  MoveL 9737 to (-47.88, -48.32, -15.5) mm, rotated rx 180 ry 0 rz 90 deg; joints [71.765, -17.653, 86.431, 0, 21.222, 71.765]
  Establecer velocidad (1000.0 mm/s)
  MoveL 9738 to (-47.88, -48.32, 10) mm, rotated rx 180 ry 0 rz 90 deg; joints [71.765, -18.97, 87.289, 0, 21.68, 71.765]
  Establecer velocidad (66.7 mm/s)
  MoveL 9739 to (-51.43, -54.96, 10) mm, rotated rx 180 ry 0 rz 90 deg; joints [71.511, -18.993, 87.381, 0, 21.611, 71.511]
  MoveL 9740 to (-51.43, -54.96, -15.5) mm, rotated rx -180 ry 0 rz 90 deg; joints [71.511, -17.675, 86.523, 0, 21.152, 71.511]
  MoveL 9741 to (-49.93, -55.15, -15.91) mm, rotated rx -180 ry 0 rz 90 deg; joints [71.521, -17.628, 86.402, 0, 21.226, 71.521]
  MoveL 9742 to (-48.42, -54.96, -16.31) mm, rotated rx -180 ry 0 rz 90 deg; joints [71.544, -17.583, 86.289, 0, 21.294, 71.544]
  MoveL 9743 to (-46.99, -54.45, -16.72) mm, rotated rx 180 ry 0 rz 90 deg; joints [71.576, -17.541, 86.189, 0, 21.352, 71.576]
  MoveL 9744 to (-45.7, -53.64, -17.12) mm, rotated rx 180 ry 0 rz 90 deg; joints [71.616, -17.504, 86.106, 0, 21.398, 71.616]
  MoveL 9745 to (-44.64, -52.56, -17.53) mm, rotated rx 180 ry 0 rz 90 deg; joints [71.663, -17.471, 86.043, 0, 21.428, 71.663]
  MoveL 9746 to (-43.83, -51.27, -17.94) mm, rotated rx -180 ry 0 rz 90 deg; joints [71.713, -17.443, 86.003, 0, 21.44, 71.713]
  MoveL 9747 to (-43.33, -49.83, -18.34) mm, rotated rx 180 ry 0 rz 90 deg; joints [71.765, -17.422, 85.987, 0, 21.435, 71.765]
  MoveL 9748 to (-43.19, -48.32, -18.75) mm, rotated rx -180 ry 0 rz 90 deg; joints [71.816, -17.407, 85.998, 0, 21.409, 71.816]
  MoveL 9749 to (-43.19, -30.36, -18.75) mm, rotated rx -180 ry 0 rz 90 deg; joints [72.401, -17.503, 86.396, 0, 21.108, 72.401]
  MoveL 9750 to (-45.96, -30.86, -18.75) mm, rotated rx -180 ry 0 rz 90 deg; joints [72.356, -17.546, 86.574, 0, 20.972, 72.356]
  MoveL 9751 to (-62.07, -33.84, -18.75) mm, rotated rx -180 ry 0 rz 90 deg; joints [72.088, -17.79, 87.605, 0, 20.185, 72.088]
  MoveL 9752 to (-65.86, -34.57, -18.75) mm, rotated rx 180 ry 0 rz 90 deg; joints [72.024, -17.845, 87.845, 0, 20.001, 72.024]
  MoveC 9753 to (-67.04, -35.24, -18.75) mm, rotated rx -180 ry 0 rz 90 deg; joints [71.989, -17.86, 87.909, 0, 19.951, 71.989] to (-67.55, -36.48, -18.75) mm, rotated rx 180 ry 0 rz 90 deg; joints [71.942, -17.862, 87.917, 0, 19.945, 71.942]
  MoveL 9754 to (-67.58, -36.96, -18.75) mm, rotated rx 180 ry 0 rz 90 deg; joints [71.926, -17.86, 87.908, 0, 19.952, 71.926]
  MoveL 9755 to (-67.57, -65.53, -18.75) mm, rotated rx 180 ry 0 rz 90 deg; joints [70.987, -17.71, 87.262, 0, 20.447, 70.987]
  MoveC 9756 to (-66.92, -67.07, -18.75) mm, rotated rx -180 ry 0 rz 90 deg; joints [70.944, -17.691, 87.182, 0, 20.509, 70.944] to (-65.35, -67.68, -18.75) mm, rotated rx -180 ry 0 rz 90 deg; joints [70.942, -17.663, 87.062, 0, 20.6, 70.942]
  MoveC 9757 to (-54.27, -67.34, -18.75) mm, rotated rx 180 ry 0 rz 90 deg; joints [71.077, -17.485, 86.319, 0, 21.166, 71.077] to (-43.19, -66.92, -18.75) mm, rotated rx 180 ry 0 rz 90 deg; joints [71.213, -17.302, 85.571, 0, 21.731, 71.213]
  MoveL 9758 to (-43.19, -48.32, -18.75) mm, rotated rx -180 ry 0 rz 90 deg; joints [71.816, -17.407, 85.998, 0, 21.409, 71.816]
  MoveL 9759 to (-50.74, -48.32, -18.75) mm, rotated rx -180 ry 0 rz 90 deg; joints [71.735, -17.532, 86.514, 0, 21.018, 71.735]
  MoveL 9760 to (-50.74, -48.32, -15.75) mm, rotated rx 180 ry 0 rz 90 deg; joints [71.735, -17.687, 86.618, 0, 21.069, 71.735]
  Establecer velocidad (1000.0 mm/s)
  MoveL 9761 to (-50.74, -48.32, 10) mm, rotated rx 180 ry 0 rz 90 deg; joints [71.735, -19.018, 87.485, 0, 21.534, 71.735]
  Establecer velocidad (66.7 mm/s)
  MoveL 9762 to (-59.34, 34.85, 10) mm, rotated rx 180 ry 0 rz 90 deg; joints [74.408, -19.568, 89.788, 0, 19.78, 74.408]
  MoveL 9763 to (-59.34, 34.85, -15.5) mm, rotated rx 180 ry 0 rz 90 deg; joints [74.408, -18.236, 88.929, 0, 19.307, 74.408]
  MoveL 9764 to (-60.84, 35.03, -15.91) mm, rotated rx 180 ry 0 rz 90 deg; joints [74.4, -18.238, 89.02, 0, 19.218, 74.4]
  MoveL 9765 to (-62.35, 34.85, -16.31) mm, rotated rx 180 ry 0 rz 90 deg; joints [74.38, -18.239, 89.104, 0, 19.135, 74.38]
  MoveL 9766 to (-63.78, 34.34, -16.72) mm, rotated rx 180 ry 0 rz 90 deg; joints [74.349, -18.237, 89.177, 0, 19.06, 74.349]
  MoveL 9767 to (-65.06, 33.52, -17.12) mm, rotated rx -180 ry 0 rz 90 deg; joints [74.309, -18.231, 89.234, 0, 18.997, 74.309]
  MoveL 9768 to (-66.13, 32.44, -17.53) mm, rotated rx -180 ry 0 rz 90 deg; joints [74.262, -18.221, 89.271, 0, 18.95, 74.262]
  MoveL 9769 to (-66.94, 31.15, -17.94) mm, rotated rx 180 ry 0 rz 90 deg; joints [74.211, -18.207, 89.287, 0, 18.92, 74.211]
  MoveL 9770 to (-67.44, 29.72, -18.34) mm, rotated rx 180 ry 0 rz 90 deg; joints [74.158, -18.187, 89.279, 0, 18.907, 74.158]
  MoveL 9771 to (-67.58, 28.21, -18.75) mm, rotated rx 180 ry 0 rz 90 deg; joints [74.105, -18.161, 89.246, 0, 18.915, 74.105]
  MoveL 9772 to (-67.58, 7.58, -18.75) mm, rotated rx 180 ry 0 rz 90 deg; joints [73.41, -18.072, 88.842, 0, 19.229, 73.41]
  MoveL 9773 to (-67.56, 7.11, -18.75) mm, rotated rx 180 ry 0 rz 90 deg; joints [73.394, -18.069, 88.832, 0, 19.237, 73.394]
  MoveC 9774 to (-66.64, 5.61, -18.75) mm, rotated rx 180 ry 0 rz 90 deg; joints [73.354, -18.049, 88.74, 0, 19.309, 73.354] to (-64.91, 5.24, -18.75) mm, rotated rx 180 ry 0 rz 90 deg; joints [73.358, -18.021, 88.616, 0, 19.405, 73.358]
  MoveL 9775 to (-63.02, 5.72, -18.75) mm, rotated rx 180 ry 0 rz 90 deg; joints [73.393, -17.994, 88.498, 0, 19.496, 73.393]
  MoveL 9776 to (-45.01, 10.34, -18.75) mm, rotated rx 180 ry 0 rz 90 deg; joints [73.724, -17.735, 87.369, 0, 20.366, 73.724]
  MoveL 9777 to (-43.19, 10.83, -18.75) mm, rotated rx 180 ry 0 rz 90 deg; joints [73.758, -17.708, 87.254, 0, 20.454, 73.758]
  MoveL 9778 to (-43.19, 36.65, -18.75) mm, rotated rx 180 ry 0 rz 90 deg; joints [74.619, -17.824, 87.754, 0, 20.07, 74.619]
  MoveC 9779 to (-53.63, 43.7, -18.75) mm, rotated rx 180 ry 0 rz 90 deg; joints [74.76, -18.017, 88.596, 0, 19.42, 74.76] to (-64.1, 50.7, -18.75) mm, rotated rx 180 ry 0 rz 90 deg; joints [74.901, -18.202, 89.431, 0, 18.771, 74.901]
  MoveC 9780 to (-64.36, 50.84, -18.75) mm, rotated rx -180 ry 0 rz 90 deg; joints [74.903, -18.206, 89.451, 0, 18.755, 74.903] to (-64.66, 50.91, -18.75) mm, rotated rx 180 ry 0 rz 90 deg; joints [74.903, -18.211, 89.472, 0, 18.739, 74.903]
  MoveC 9781 to (-66.38, 50.6, -18.75) mm, rotated rx 180 ry 0 rz 90 deg; joints [74.876, -18.235, 89.583, 0, 18.652, 74.876] to (-67.57, 49.31, -18.75) mm, rotated rx 180 ry 0 rz 90 deg; joints [74.822, -18.247, 89.639, 0, 18.608, 74.822]
  MoveL 9782 to (-67.58, 48.8, -18.75) mm, rotated rx -180 ry 0 rz 90 deg; joints [74.804, -18.245, 89.63, 0, 18.615, 74.804]
  MoveL 9783 to (-67.58, 28.21, -18.75) mm, rotated rx 180 ry 0 rz 90 deg; joints [74.105, -18.161, 89.246, 0, 18.915, 74.105]
  MoveL 9784 to (-60.03, 28.21, -18.75) mm, rotated rx -180 ry 0 rz 90 deg; joints [74.178, -18.048, 88.738, 0, 19.311, 74.178]
  MoveL 9785 to (-60.03, 28.21, -15.75) mm, rotated rx 180 ry 0 rz 90 deg; joints [74.178, -18.205, 88.841, 0, 19.364, 74.178]
  Establecer velocidad (1000.0 mm/s)
  MoveL 9786 to (-60.03, 28.21, 10) mm, rotated rx -180 ry 0 rz 90 deg; joints [74.178, -19.549, 89.708, 0, 19.841, 74.178]
  Establecer velocidad (66.7 mm/s)
  MoveL 9787 to (-59.17, 34.85, 10) mm, rotated rx 180 ry 0 rz 90 deg; joints [74.41, -19.565, 89.777, 0, 19.789, 74.41]
  MoveL 9788 to (-59.17, 34.85, -15.75) mm, rotated rx 180 ry 0 rz 90 deg; joints [74.41, -18.22, 88.909, 0, 19.311, 74.41]
  MoveL 9789 to (-60.68, 35.03, -16.16) mm, rotated rx 180 ry 0 rz 90 deg; joints [74.402, -18.223, 89, 0, 19.222, 74.402]
  MoveL 9790 to (-62.19, 34.85, -16.56) mm, rotated rx 180 ry 0 rz 90 deg; joints [74.381, -18.223, 89.085, 0, 19.139, 74.381]
  MoveL 9791 to (-63.62, 34.34, -16.97) mm, rotated rx -180 ry 0 rz 90 deg; joints [74.351, -18.221, 89.158, 0, 19.064, 74.351]
  MoveL 9792 to (-64.9, 33.52, -17.38) mm, rotated rx 180 ry 0 rz 90 deg; joints [74.311, -18.216, 89.214, 0, 19.002, 74.311]
  MoveL 9793 to (-65.97, 32.44, -17.78) mm, rotated rx 180 ry 0 rz 90 deg; joints [74.264, -18.206, 89.252, 0, 18.954, 74.264]
  MoveL 9794 to (-66.77, 31.15, -18.19) mm, rotated rx 180 ry 0 rz 90 deg; joints [74.213, -18.191, 89.267, 0, 18.924, 74.213]
  MoveL 9795 to (-67.27, 29.72, -18.59) mm, rotated rx 180 ry 0 rz 90 deg; joints [74.159, -18.171, 89.26, 0, 18.912, 74.159]
  MoveL 9796 to (-67.41, 28.21, -19) mm, rotated rx 180 ry 0 rz 90 deg; joints [74.107, -18.146, 89.226, 0, 18.92, 74.107]
  MoveL 9797 to (-67.41, 7.58, -19) mm, rotated rx 180 ry 0 rz 90 deg; joints [73.412, -18.056, 88.823, 0, 19.234, 73.412]
  MoveC 9798 to (-66.67, 5.91, -19) mm, rotated rx 180 ry 0 rz 90 deg; joints [73.363, -18.038, 88.739, 0, 19.298, 73.363] to (-64.91, 5.4, -19) mm, rotated rx 180 ry 0 rz 90 deg; joints [73.364, -18.009, 88.611, 0, 19.398, 73.364]
  MoveL 9799 to (-64.44, 5.5, -19) mm, rotated rx -180 ry 0 rz 90 deg; joints [73.372, -18.002, 88.581, 0, 19.421, 73.372]
  MoveL 9800 to (-61.12, 6.33, -19) mm, rotated rx 180 ry 0 rz 90 deg; joints [73.433, -17.955, 88.374, 0, 19.581, 73.433]
  MoveL 9801 to (-46.91, 10, -19) mm, rotated rx 180 ry 0 rz 90 deg; joints [73.695, -17.75, 87.483, 0, 20.267, 73.695]
  MoveL 9802 to (-46.05, 10.22, -19) mm, rotated rx 180 ry 0 rz 90 deg; joints [73.711, -17.738, 87.429, 0, 20.309, 73.711]
  MoveL 9803 to (-46.05, 38.41, -19) mm, rotated rx -180 ry 0 rz 90 deg; joints [74.652, -17.864, 87.974, 0, 19.89, 74.652]
  MoveC 9804 to (-55.14, 44.54, -19) mm, rotated rx 180 ry 0 rz 90 deg; joints [74.775, -18.03, 88.705, 0, 19.325, 74.775] to (-64.26, 50.63, -19) mm, rotated rx -180 ry 0 rz 90 deg; joints [74.897, -18.191, 89.432, 0, 18.759, 74.897]
  MoveC 9805 to (-66.11, 50.42, -19) mm, rotated rx 180 ry 0 rz 90 deg; joints [74.873, -18.217, 89.552, 0, 18.665, 74.873] to (-67.41, 49.08, -19) mm, rotated rx -180 ry 0 rz 90 deg; joints [74.815, -18.231, 89.615, 0, 18.616, 74.815]
  MoveL 9806 to (-67.41, 48.8, -19) mm, rotated rx -180 ry 0 rz 90 deg; joints [74.806, -18.23, 89.611, 0, 18.619, 74.806]
  MoveL 9807 to (-67.41, 28.21, -19) mm, rotated rx 180 ry 0 rz 90 deg; joints [74.107, -18.146, 89.226, 0, 18.92, 74.107]
  MoveL 9808 to (-59.86, 28.21, -19) mm, rotated rx 180 ry 0 rz 90 deg; joints [74.179, -18.033, 88.718, 0, 19.315, 74.179]
  MoveL 9809 to (-59.86, 28.21, -16) mm, rotated rx 180 ry 0 rz 90 deg; joints [74.179, -18.19, 88.821, 0, 19.368, 74.179]
  Establecer velocidad (1000.0 mm/s)
  MoveL 9810 to (-59.86, 28.21, 10) mm, rotated rx 180 ry 0 rz 90 deg; joints [74.179, -19.547, 89.697, 0, 19.85, 74.179]
  Establecer velocidad (66.7 mm/s)
  MoveL 9811 to (-59.17, -44.43, 10) mm, rotated rx -180 ry 0 rz 90 deg; joints [71.771, -19.18, 88.145, 0, 21.035, 71.771]
  MoveL 9812 to (-59.17, -44.43, -15.75) mm, rotated rx 180 ry 0 rz 90 deg; joints [71.771, -17.845, 87.278, 0, 20.567, 71.771]
  MoveL 9813 to (-60.68, -44.25, -16.16) mm, rotated rx 180 ry 0 rz 90 deg; joints [71.761, -17.849, 87.37, 0, 20.478, 71.761]
  MoveL 9814 to (-62.19, -44.43, -16.56) mm, rotated rx 180 ry 0 rz 90 deg; joints [71.738, -17.851, 87.454, 0, 20.396, 71.738]
  MoveL 9815 to (-63.62, -44.94, -16.97) mm, rotated rx 180 ry 0 rz 90 deg; joints [71.706, -17.85, 87.526, 0, 20.324, 71.706]
  MoveL 9816 to (-64.9, -45.76, -17.38) mm, rotated rx -180 ry 0 rz 90 deg; joints [71.665, -17.844, 87.58, 0, 20.264, 71.665]
  MoveL 9817 to (-65.97, -46.84, -17.78) mm, rotated rx -180 ry 0 rz 90 deg; joints [71.618, -17.835, 87.614, 0, 20.221, 71.618]
  MoveL 9818 to (-66.77, -48.13, -18.19) mm, rotated rx -180 ry 0 rz 90 deg; joints [71.567, -17.819, 87.625, 0, 20.194, 71.567]
  MoveL 9819 to (-67.27, -49.56, -18.59) mm, rotated rx -180 ry 0 rz 90 deg; joints [71.514, -17.798, 87.613, 0, 20.186, 71.514]
  MoveL 9820 to (-67.41, -51.07, -19) mm, rotated rx 180 ry 0 rz 90 deg; joints [71.463, -17.772, 87.574, 0, 20.198, 71.463]
  MoveL 9821 to (-67.41, -64.91, -19) mm, rotated rx 180 ry 0 rz 90 deg; joints [71.009, -17.698, 87.257, 0, 20.44, 71.009]
  MoveL 9822 to (-67.41, -65.39, -19) mm, rotated rx -180 ry 0 rz 90 deg; joints [70.994, -17.695, 87.246, 0, 20.449, 70.994]
  MoveC 9823 to (-66.84, -66.87, -19) mm, rotated rx 180 ry 0 rz 90 deg; joints [70.952, -17.678, 87.173, 0, 20.505, 70.952] to (-65.39, -67.53, -19) mm, rotated rx -180 ry 0 rz 90 deg; joints [70.947, -17.651, 87.06, 0, 20.591, 70.947]
  MoveL 9824 to (-64.91, -67.53, -19) mm, rotated rx 180 ry 0 rz 90 deg; joints [70.952, -17.643, 87.028, 0, 20.616, 70.952]
  MoveL 9825 to (-47.86, -66.96, -19) mm, rotated rx -180 ry 0 rz 90 deg; joints [71.161, -17.368, 85.881, 0, 21.486, 71.161]
  MoveL 9826 to (-46.05, -66.87, -19) mm, rotated rx -180 ry 0 rz 90 deg; joints [71.183, -17.338, 85.759, 0, 21.578, 71.183]
  MoveL 9827 to (-46.05, -31.04, -19) mm, rotated rx -180 ry 0 rz 90 deg; joints [72.349, -17.534, 86.568, 0, 20.966, 72.349]
  MoveL 9828 to (-62.07, -34, -19) mm, rotated rx 180 ry 0 rz 90 deg; joints [72.083, -17.776, 87.593, 0, 20.183, 72.083]
  MoveL 9829 to (-65.71, -34.69, -19) mm, rotated rx -180 ry 0 rz 90 deg; joints [72.021, -17.829, 87.823, 0, 20.006, 72.021]
  MoveC 9830 to (-66.93, -35.42, -19) mm, rotated rx 180 ry 0 rz 90 deg; joints [71.984, -17.845, 87.89, 0, 19.955, 71.984] to (-67.41, -36.76, -19) mm, rotated rx -180 ry 0 rz 90 deg; joints [71.935, -17.845, 87.893, 0, 19.953, 71.935]
  MoveL 9831 to (-67.41, -51.07, -19) mm, rotated rx 180 ry 0 rz 90 deg; joints [71.463, -17.772, 87.574, 0, 20.198, 71.463]
  MoveL 9832 to (-59.86, -51.07, -19) mm, rotated rx -180 ry 0 rz 90 deg; joints [71.546, -17.652, 87.064, 0, 20.588, 71.546]
  MoveL 9833 to (-59.86, -51.07, -16) mm, rotated rx 180 ry 0 rz 90 deg; joints [71.546, -17.808, 87.167, 0, 20.64, 71.546]
  Establecer velocidad (1000.0 mm/s)
  MoveL 9834 to (-59.86, -51.07, 10) mm, rotated rx -180 ry 0 rz 90 deg; joints [71.546, -19.155, 88.042, 0, 21.112, 71.546]
  Establecer velocidad (66.7 mm/s)
  MoveL 9835 to (-59.01, -44.43, 10) mm, rotated rx 180 ry 0 rz 90 deg; joints [71.773, -19.177, 88.134, 0, 21.043, 71.773]
  MoveL 9836 to (-59.01, -44.43, -16) mm, rotated rx 180 ry 0 rz 90 deg; joints [71.773, -17.829, 87.259, 0, 20.571, 71.773]
  MoveL 9837 to (-60.51, -44.25, -16.41) mm, rotated rx 180 ry 0 rz 90 deg; joints [71.762, -17.833, 87.351, 0, 20.483, 71.762]
  MoveL 9838 to (-62.02, -44.43, -16.81) mm, rotated rx 180 ry 0 rz 90 deg; joints [71.74, -17.835, 87.435, 0, 20.401, 71.74]
  MoveL 9839 to (-63.45, -44.94, -17.22) mm, rotated rx -180 ry 0 rz 90 deg; joints [71.708, -17.834, 87.506, 0, 20.328, 71.708]
  MoveL 9840 to (-64.73, -45.76, -17.63) mm, rotated rx -180 ry 0 rz 90 deg; joints [71.667, -17.829, 87.56, 0, 20.269, 71.667]
  MoveL 9841 to (-65.81, -46.84, -18.03) mm, rotated rx 180 ry 0 rz 90 deg; joints [71.62, -17.819, 87.594, 0, 20.225, 71.62]
  MoveL 9842 to (-66.61, -48.13, -18.44) mm, rotated rx -180 ry 0 rz 90 deg; joints [71.569, -17.804, 87.605, 0, 20.198, 71.569]
  MoveL 9843 to (-67.11, -49.56, -18.84) mm, rotated rx -180 ry 0 rz 90 deg; joints [71.516, -17.783, 87.593, 0, 20.19, 71.516]
  MoveL 9844 to (-67.25, -51.07, -19.25) mm, rotated rx 180 ry 0 rz 90 deg; joints [71.465, -17.756, 87.554, 0, 20.202, 71.465]
  MoveL 9845 to (-67.25, -65.29, -19.25) mm, rotated rx -180 ry 0 rz 90 deg; joints [70.999, -17.68, 87.229, 0, 20.451, 70.999]
  MoveC 9846 to (-66.61, -66.8, -19.25) mm, rotated rx 180 ry 0 rz 90 deg; joints [70.957, -17.661, 87.15, 0, 20.511, 70.957] to (-65.07, -67.4, -19.25) mm, rotated rx -180 ry 0 rz 90 deg; joints [70.955, -17.634, 87.033, 0, 20.601, 70.955]
  MoveL 9847 to (-63.02, -67.33, -19.25) mm, rotated rx 180 ry 0 rz 90 deg; joints [70.98, -17.601, 86.895, 0, 20.706, 70.98]
  MoveL 9848 to (-51.65, -66.94, -19.25) mm, rotated rx -180 ry 0 rz 90 deg; joints [71.119, -17.418, 86.132, 0, 21.286, 71.119]
  MoveL 9849 to (-48.91, -66.84, -19.25) mm, rotated rx -180 ry 0 rz 90 deg; joints [71.153, -17.373, 85.947, 0, 21.426, 71.153]
  MoveL 9850 to (-48.91, -31.73, -19.25) mm, rotated rx 180 ry 0 rz 90 deg; joints [72.297, -17.564, 86.74, 0, 20.824, 72.297]
  MoveL 9851 to (-51.65, -32.22, -19.25) mm, rotated rx -180 ry 0 rz 90 deg; joints [72.252, -17.606, 86.916, 0, 20.69, 72.252]
  MoveL 9852 to (-65.58, -34.82, -19.25) mm, rotated rx 180 ry 0 rz 90 deg; joints [72.019, -17.814, 87.803, 0, 20.011, 72.019]
  MoveC 9853 to (-66.78, -35.52, -19.25) mm, rotated rx 180 ry 0 rz 90 deg; joints [71.983, -17.829, 87.868, 0, 19.961, 71.983] to (-67.25, -36.82, -19.25) mm, rotated rx -180 ry 0 rz 90 deg; joints [71.934, -17.829, 87.871, 0, 19.958, 71.934]
  MoveL 9854 to (-67.25, -51.07, -19.25) mm, rotated rx 180 ry 0 rz 90 deg; joints [71.465, -17.756, 87.554, 0, 20.202, 71.465]
  MoveL 9855 to (-59.7, -51.07, -19.25) mm, rotated rx -180 ry 0 rz 90 deg; joints [71.548, -17.636, 87.044, 0, 20.592, 71.548]
  MoveL 9856 to (-59.7, -51.07, -16.25) mm, rotated rx 180 ry 0 rz 90 deg; joints [71.548, -17.792, 87.147, 0, 20.645, 71.548]
  Establecer velocidad (1000.0 mm/s)
  MoveL 9857 to (-59.7, -51.07, 10) mm, rotated rx 180 ry 0 rz 90 deg; joints [71.548, -19.152, 88.031, 0, 21.121, 71.548]
  Establecer velocidad (66.7 mm/s)
  MoveL 9858 to (-59.01, 34.87, 10) mm, rotated rx -180 ry 0 rz 90 deg; joints [74.412, -19.563, 89.766, 0, 19.797, 74.412]
  MoveL 9859 to (-59.01, 34.87, -16) mm, rotated rx 180 ry 0 rz 90 deg; joints [74.412, -18.205, 88.89, 0, 19.315, 74.412]
  MoveL 9860 to (-60.52, 35.05, -16.41) mm, rotated rx 180 ry 0 rz 90 deg; joints [74.404, -18.207, 88.981, 0, 19.226, 74.404]
  MoveL 9861 to (-62.02, 34.87, -16.81) mm, rotated rx -180 ry 0 rz 90 deg; joints [74.384, -18.208, 89.066, 0, 19.142, 74.384]
  MoveL 9862 to (-63.45, 34.36, -17.22) mm, rotated rx -180 ry 0 rz 90 deg; joints [74.353, -18.206, 89.138, 0, 19.068, 74.353]
  MoveL 9863 to (-64.74, 33.54, -17.63) mm, rotated rx 180 ry 0 rz 90 deg; joints [74.313, -18.2, 89.195, 0, 19.005, 74.313]
  MoveL 9864 to (-65.81, 32.46, -18.03) mm, rotated rx -180 ry 0 rz 90 deg; joints [74.266, -18.19, 89.233, 0, 18.958, 74.266]
  MoveL 9865 to (-66.61, 31.18, -18.44) mm, rotated rx -180 ry 0 rz 90 deg; joints [74.215, -18.176, 89.248, 0, 18.927, 74.215]
  MoveL 9866 to (-67.11, 29.74, -18.84) mm, rotated rx 180 ry 0 rz 90 deg; joints [74.162, -18.156, 89.24, 0, 18.915, 74.162]
  MoveL 9867 to (-67.25, 28.23, -19.25) mm, rotated rx -180 ry 0 rz 90 deg; joints [74.109, -18.13, 89.207, 0, 18.923, 74.109]
  MoveL 9868 to (-67.25, 8.05, -19.25) mm, rotated rx 180 ry 0 rz 90 deg; joints [73.429, -18.043, 88.812, 0, 19.23, 73.429]
  MoveL 9869 to (-67.25, 7.58, -19.25) mm, rotated rx 180 ry 0 rz 90 deg; joints [73.414, -18.041, 88.803, 0, 19.238, 73.414]
  MoveC 9870 to (-66.51, 6.08, -19.25) mm, rotated rx 180 ry 0 rz 90 deg; joints [73.37, -18.023, 88.723, 0, 19.3, 73.37] to (-64.91, 5.55, -19.25) mm, rotated rx 180 ry 0 rz 90 deg; joints [73.369, -17.996, 88.605, 0, 19.391, 73.369]
  MoveL 9871 to (-64.44, 5.64, -19.25) mm, rotated rx 180 ry 0 rz 90 deg; joints [73.377, -17.99, 88.575, 0, 19.414, 73.377]
  MoveL 9872 to (-48.91, 9.64, -19.25) mm, rotated rx -180 ry 0 rz 90 deg; joints [73.663, -17.767, 87.603, 0, 20.164, 73.663]
  MoveL 9873 to (-48.91, 40.16, -19.25) mm, rotated rx 180 ry 0 rz 90 deg; joints [74.684, -17.903, 88.192, 0, 19.71, 74.684]
  MoveL 9874 to (-60.32, 47.86, -19.25) mm, rotated rx 180 ry 0 rz 90 deg; joints [74.839, -18.108, 89.107, 0, 19.001, 74.839]
  MoveL 9875 to (-63.15, 49.75, -19.25) mm, rotated rx 180 ry 0 rz 90 deg; joints [74.877, -18.158, 89.333, 0, 18.825, 74.877]
  MoveL 9876 to (-63.97, 50.3, -19.25) mm, rotated rx -180 ry 0 rz 90 deg; joints [74.888, -18.172, 89.398, 0, 18.775, 74.888]
  MoveL 9877 to (-64.12, 50.38, -19.25) mm, rotated rx 180 ry 0 rz 90 deg; joints [74.89, -18.175, 89.41, 0, 18.765, 74.89]
  MoveC 9878 to (-65.95, 50.18, -19.25) mm, rotated rx 180 ry 0 rz 90 deg; joints [74.866, -18.201, 89.528, 0, 18.672, 74.866] to (-67.24, 48.88, -19.25) mm, rotated rx -180 ry 0 rz 90 deg; joints [74.81, -18.214, 89.592, 0, 18.623, 74.81]
  MoveL 9879 to (-67.25, 48.8, -19.25) mm, rotated rx -180 ry 0 rz 90 deg; joints [74.807, -18.214, 89.591, 0, 18.623, 74.807]
  MoveL 9880 to (-67.25, 28.23, -19.25) mm, rotated rx -180 ry 0 rz 90 deg; joints [74.109, -18.13, 89.207, 0, 18.923, 74.109]
  MoveL 9881 to (-59.7, 28.23, -19.25) mm, rotated rx -180 ry 0 rz 90 deg; joints [74.182, -18.017, 88.698, 0, 19.319, 74.182]
  MoveL 9882 to (-59.7, 28.23, -16.25) mm, rotated rx 180 ry 0 rz 90 deg; joints [74.182, -18.174, 88.802, 0, 19.372, 74.182]
  Establecer velocidad (1000.0 mm/s)
  MoveL 9883 to (-59.7, 28.23, 10) mm, rotated rx 180 ry 0 rz 90 deg; joints [74.182, -19.544, 89.686, 0, 19.858, 74.182]
  Establecer velocidad (66.7 mm/s)
  MoveL 9884 to (-58.84, 34.87, 10) mm, rotated rx -180 ry 0 rz 90 deg; joints [74.414, -19.56, 89.755, 0, 19.805, 74.414]
  MoveL 9885 to (-58.84, 34.87, -16.25) mm, rotated rx 180 ry 0 rz 90 deg; joints [74.414, -18.189, 88.87, 0, 19.319, 74.414]
  MoveL 9886 to (-60.35, 35.05, -16.66) mm, rotated rx 180 ry 0 rz 90 deg; joints [74.406, -18.192, 88.962, 0, 19.23, 74.406]
  MoveL 9887 to (-61.86, 34.87, -17.06) mm, rotated rx -180 ry 0 rz 90 deg; joints [74.385, -18.192, 89.046, 0, 19.147, 74.385]
  MoveL 9888 to (-63.29, 34.36, -17.47) mm, rotated rx -180 ry 0 rz 90 deg; joints [74.354, -18.19, 89.119, 0, 19.072, 74.354]
  MoveL 9889 to (-64.57, 33.54, -17.87) mm, rotated rx -180 ry 0 rz 90 deg; joints [74.315, -18.185, 89.175, 0, 19.009, 74.315]
  MoveL 9890 to (-65.64, 32.46, -18.28) mm, rotated rx -180 ry 0 rz 90 deg; joints [74.268, -18.175, 89.213, 0, 18.962, 74.268]
  MoveL 9891 to (-66.45, 31.18, -18.69) mm, rotated rx -180 ry 0 rz 90 deg; joints [74.217, -18.16, 89.229, 0, 18.932, 74.217]
  MoveL 9892 to (-66.94, 29.74, -19.09) mm, rotated rx 180 ry 0 rz 90 deg; joints [74.163, -18.14, 89.221, 0, 18.92, 74.163]
  MoveL 9893 to (-67.08, 28.23, -19.5) mm, rotated rx 180 ry 0 rz 90 deg; joints [74.111, -18.115, 89.187, 0, 18.928, 74.111]
  MoveL 9894 to (-67.08, 8.05, -19.5) mm, rotated rx -180 ry 0 rz 90 deg; joints [73.431, -18.027, 88.793, 0, 19.235, 73.431]
  MoveL 9895 to (-67.07, 7.58, -19.5) mm, rotated rx -180 ry 0 rz 90 deg; joints [73.415, -18.025, 88.783, 0, 19.242, 73.415]
  MoveC 9896 to (-66.15, 6.1, -19.5) mm, rotated rx 180 ry 0 rz 90 deg; joints [73.375, -18.005, 88.691, 0, 19.313, 73.375] to (-64.44, 5.79, -19.5) mm, rotated rx -180 ry 0 rz 90 deg; joints [73.381, -17.977, 88.57, 0, 19.408, 73.381]
  MoveL 9897 to (-51.77, 9.04, -19.5) mm, rotated rx 180 ry 0 rz 90 deg; joints [73.616, -17.797, 87.777, 0, 20.019, 73.616]
  MoveL 9898 to (-51.77, 41.93, -19.5) mm, rotated rx 180 ry 0 rz 90 deg; joints [74.718, -17.941, 88.411, 0, 19.53, 74.718]
  MoveL 9899 to (-53.54, 43.14, -19.5) mm, rotated rx -180 ry 0 rz 90 deg; joints [74.742, -17.974, 88.554, 0, 19.42, 74.742]
  MoveL 9900 to (-63.49, 49.82, -19.5) mm, rotated rx -180 ry 0 rz 90 deg; joints [74.877, -18.15, 89.348, 0, 18.802, 74.877]
  MoveL 9901 to (-63.97, 50.13, -19.5) mm, rotated rx -180 ry 0 rz 90 deg; joints [74.883, -18.158, 89.386, 0, 18.772, 74.883]
  MoveC 9902 to (-65.78, 49.95, -19.5) mm, rotated rx 180 ry 0 rz 90 deg; joints [74.86, -18.184, 89.505, 0, 18.68, 74.86] to (-67.08, 48.67, -19.5) mm, rotated rx 180 ry 0 rz 90 deg; joints [74.804, -18.198, 89.569, 0, 18.63, 74.804]
  MoveL 9903 to (-67.08, 28.23, -19.5) mm, rotated rx 180 ry 0 rz 90 deg; joints [74.111, -18.115, 89.187, 0, 18.928, 74.111]
  MoveL 9904 to (-59.54, 28.23, -19.5) mm, rotated rx -180 ry 0 rz 90 deg; joints [74.183, -18.002, 88.679, 0, 19.323, 74.183]
  MoveL 9905 to (-59.54, 28.23, -16.5) mm, rotated rx -180 ry 0 rz 90 deg; joints [74.183, -18.159, 88.782, 0, 19.376, 74.183]
  Establecer velocidad (1000.0 mm/s)
  MoveL 9906 to (-59.54, 28.23, 10) mm, rotated rx -180 ry 0 rz 90 deg; joints [74.183, -19.542, 89.675, 0, 19.867, 74.183]
  Establecer velocidad (66.7 mm/s)
  MoveL 9907 to (-58.84, -44.46, 10) mm, rotated rx 180 ry 0 rz 90 deg; joints [71.774, -19.174, 88.122, 0, 21.052, 71.774]
  MoveL 9908 to (-58.84, -44.46, -16.25) mm, rotated rx 180 ry 0 rz 90 deg; joints [71.774, -17.813, 87.238, 0, 20.575, 71.774]
  MoveL 9909 to (-60.35, -44.27, -16.66) mm, rotated rx -180 ry 0 rz 90 deg; joints [71.763, -17.817, 87.33, 0, 20.487, 71.763]
  MoveL 9910 to (-61.86, -44.46, -17.06) mm, rotated rx 180 ry 0 rz 90 deg; joints [71.741, -17.819, 87.414, 0, 20.405, 71.741]
  MoveL 9911 to (-63.29, -44.97, -17.47) mm, rotated rx 180 ry 0 rz 90 deg; joints [71.709, -17.818, 87.486, 0, 20.333, 71.709]
  MoveL 9912 to (-64.57, -45.79, -17.87) mm, rotated rx -180 ry 0 rz 90 deg; joints [71.668, -17.813, 87.54, 0, 20.273, 71.668]
  MoveL 9913 to (-65.64, -46.87, -18.28) mm, rotated rx -180 ry 0 rz 90 deg; joints [71.621, -17.803, 87.574, 0, 20.229, 71.621]
  MoveL 9914 to (-66.45, -48.15, -18.69) mm, rotated rx -180 ry 0 rz 90 deg; joints [71.57, -17.788, 87.585, 0, 20.203, 71.57]
  MoveL 9915 to (-66.94, -49.59, -19.09) mm, rotated rx -180 ry 0 rz 90 deg; joints [71.517, -17.767, 87.572, 0, 20.195, 71.517]
  MoveL 9916 to (-67.08, -51.1, -19.5) mm, rotated rx 180 ry 0 rz 90 deg; joints [71.466, -17.74, 87.534, 0, 20.206, 71.466]
  MoveL 9917 to (-67.08, -64.91, -19.5) mm, rotated rx 180 ry 0 rz 90 deg; joints [71.013, -17.666, 87.218, 0, 20.449, 71.013]
  MoveL 9918 to (-67.07, -65.24, -19.5) mm, rotated rx 180 ry 0 rz 90 deg; joints [71.002, -17.664, 87.209, 0, 20.455, 71.002]
  MoveC 9919 to (-66.43, -66.68, -19.5) mm, rotated rx 180 ry 0 rz 90 deg; joints [70.963, -17.646, 87.132, 0, 20.514, 70.963] to (-64.95, -67.25, -19.5) mm, rotated rx -180 ry 0 rz 90 deg; joints [70.961, -17.62, 87.02, 0, 20.6, 70.961]
  MoveL 9920 to (-63.97, -67.22, -19.5) mm, rotated rx -180 ry 0 rz 90 deg; joints [70.973, -17.604, 86.954, 0, 20.65, 70.973]
  MoveL 9921 to (-51.77, -66.79, -19.5) mm, rotated rx -180 ry 0 rz 90 deg; joints [71.123, -17.408, 86.135, 0, 21.273, 71.123]
  MoveL 9922 to (-51.77, -32.4, -19.5) mm, rotated rx 180 ry 0 rz 90 deg; joints [72.245, -17.594, 86.911, 0, 20.683, 72.245]
  MoveL 9923 to (-65.39, -34.93, -19.5) mm, rotated rx 180 ry 0 rz 90 deg; joints [72.017, -17.797, 87.779, 0, 20.018, 72.017]
  MoveC 9924 to (-66.61, -35.63, -19.5) mm, rotated rx 180 ry 0 rz 90 deg; joints [71.981, -17.813, 87.846, 0, 19.967, 71.981] to (-67.08, -36.96, -19.5) mm, rotated rx 180 ry 0 rz 90 deg; joints [71.932, -17.813, 87.848, 0, 19.965, 71.932]
  MoveL 9925 to (-67.08, -37.43, -19.5) mm, rotated rx 180 ry 0 rz 90 deg; joints [71.916, -17.811, 87.838, 0, 19.972, 71.916]
  MoveL 9926 to (-67.08, -51.1, -19.5) mm, rotated rx 180 ry 0 rz 90 deg; joints [71.466, -17.74, 87.534, 0, 20.206, 71.466]
  MoveL 9927 to (-59.54, -51.1, -19.5) mm, rotated rx 180 ry 0 rz 90 deg; joints [71.549, -17.621, 87.024, 0, 20.597, 71.549]
  MoveL 9928 to (-59.54, -51.1, -16.5) mm, rotated rx -180 ry 0 rz 90 deg; joints [71.549, -17.776, 87.127, 0, 20.649, 71.549]
  Establecer velocidad (1000.0 mm/s)
  MoveL 9929 to (-59.54, -51.1, 10) mm, rotated rx 180 ry 0 rz 90 deg; joints [71.549, -19.149, 88.02, 0, 21.129, 71.549]
  Establecer velocidad (66.7 mm/s)
  MoveL 9930 to (-58.32, -45.63, 10) mm, rotated rx 180 ry 0 rz 90 deg; joints [71.741, -19.159, 88.06, 0, 21.099, 71.741]
  MoveL 9931 to (-58.32, -45.63, -16.5) mm, rotated rx 180 ry 0 rz 90 deg; joints [71.741, -17.786, 87.168, 0, 20.618, 71.741]
  MoveL 9932 to (-59.76, -45.14, -16.91) mm, rotated rx 180 ry 0 rz 90 deg; joints [71.742, -17.79, 87.262, 0, 20.528, 71.742]
  MoveL 9933 to (-61.27, -45.04, -17.31) mm, rotated rx -180 ry 0 rz 90 deg; joints [71.728, -17.794, 87.353, 0, 20.441, 71.728]
  MoveL 9934 to (-62.76, -45.33, -17.72) mm, rotated rx 180 ry 0 rz 90 deg; joints [71.703, -17.795, 87.433, 0, 20.362, 71.703]
  MoveL 9935 to (-64.14, -45.98, -18.13) mm, rotated rx 180 ry 0 rz 90 deg; joints [71.666, -17.792, 87.498, 0, 20.295, 71.666]
  MoveL 9936 to (-65.31, -46.95, -18.53) mm, rotated rx -180 ry 0 rz 90 deg; joints [71.622, -17.784, 87.541, 0, 20.244, 71.622]
  MoveL 9937 to (-66.2, -48.18, -18.94) mm, rotated rx 180 ry 0 rz 90 deg; joints [71.571, -17.771, 87.559, 0, 20.211, 71.571]
  MoveL 9938 to (-66.76, -49.59, -19.34) mm, rotated rx -180 ry 0 rz 90 deg; joints [71.519, -17.751, 87.551, 0, 20.2, 71.519]
  MoveL 9939 to (-66.92, -51.1, -19.75) mm, rotated rx 180 ry 0 rz 90 deg; joints [71.468, -17.725, 87.514, 0, 20.211, 71.468]
  MoveL 9940 to (-66.92, -65.05, -19.75) mm, rotated rx 180 ry 0 rz 90 deg; joints [71.01, -17.65, 87.195, 0, 20.455, 71.01]
  MoveC 9941 to (-66.31, -66.51, -19.75) mm, rotated rx 180 ry 0 rz 90 deg; joints [70.97, -17.632, 87.119, 0, 20.513, 70.97] to (-64.83, -67.09, -19.75) mm, rotated rx -180 ry 0 rz 90 deg; joints [70.967, -17.606, 87.006, 0, 20.599, 70.967]
  MoveL 9942 to (-63.97, -67.08, -19.75) mm, rotated rx 180 ry 0 rz 90 deg; joints [70.977, -17.592, 86.948, 0, 20.644, 70.977]
  MoveL 9943 to (-54.62, -66.75, -19.75) mm, rotated rx 180 ry 0 rz 90 deg; joints [71.093, -17.442, 86.322, 0, 21.12, 71.093]
  MoveL 9944 to (-54.62, -33.08, -19.75) mm, rotated rx -180 ry 0 rz 90 deg; joints [72.192, -17.623, 87.082, 0, 20.541, 72.192]
  MoveL 9945 to (-64.91, -34.99, -19.75) mm, rotated rx 180 ry 0 rz 90 deg; joints [72.02, -17.776, 87.737, 0, 20.039, 72.02]
  MoveL 9946 to (-65.29, -35.06, -19.75) mm, rotated rx 180 ry 0 rz 90 deg; joints [72.014, -17.782, 87.761, 0, 20.021, 72.014]
  MoveC 9947 to (-66.44, -35.72, -19.75) mm, rotated rx 180 ry 0 rz 90 deg; joints [71.979, -17.796, 87.824, 0, 19.973, 71.979] to (-66.91, -36.96, -19.75) mm, rotated rx -180 ry 0 rz 90 deg; joints [71.934, -17.797, 87.828, 0, 19.969, 71.934]
  MoveL 9948 to (-66.92, -37.43, -19.75) mm, rotated rx 180 ry 0 rz 90 deg; joints [71.918, -17.795, 87.819, 0, 19.977, 71.918]
  MoveL 9949 to (-66.92, -51.1, -19.75) mm, rotated rx 180 ry 0 rz 90 deg; joints [71.468, -17.725, 87.514, 0, 20.211, 71.468]
  MoveL 9950 to (-59.37, -51.1, -19.75) mm, rotated rx -180 ry 0 rz 90 deg; joints [71.55, -17.605, 87.004, 0, 20.601, 71.55]
  MoveL 9951 to (-59.37, -51.1, -16.75) mm, rotated rx -180 ry 0 rz 90 deg; joints [71.55, -17.761, 87.107, 0, 20.653, 71.55]
  Establecer velocidad (1000.0 mm/s)
  MoveL 9952 to (-59.37, -51.1, 10) mm, rotated rx -180 ry 0 rz 90 deg; joints [71.55, -19.146, 88.009, 0, 21.138, 71.55]
  Establecer velocidad (66.7 mm/s)
  MoveL 9953 to (-58.32, 33.48, 10) mm, rotated rx 180 ry 0 rz 90 deg; joints [74.372, -19.546, 89.693, 0, 19.853, 74.372]
  MoveL 9954 to (-58.32, 33.48, -16.5) mm, rotated rx 180 ry 0 rz 90 deg; joints [74.372, -18.163, 88.8, 0, 19.362, 74.372]
  MoveL 9955 to (-59.76, 33.97, -16.91) mm, rotated rx 180 ry 0 rz 90 deg; joints [74.375, -18.165, 88.892, 0, 19.273, 74.375]
  MoveL 9956 to (-61.27, 34.06, -17.31) mm, rotated rx 180 ry 0 rz 90 deg; joints [74.363, -18.167, 88.982, 0, 19.185, 74.363]
  MoveL 9957 to (-62.77, 33.77, -17.72) mm, rotated rx 180 ry 0 rz 90 deg; joints [74.34, -18.167, 89.064, 0, 19.103, 74.34]
  MoveL 9958 to (-64.14, 33.13, -18.13) mm, rotated rx -180 ry 0 rz 90 deg; joints [74.305, -18.164, 89.13, 0, 19.034, 74.305]
  MoveL 9959 to (-65.31, 32.16, -18.53) mm, rotated rx 180 ry 0 rz 90 deg; joints [74.261, -18.156, 89.176, 0, 18.98, 74.261]
  MoveL 9960 to (-66.2, 30.93, -18.94) mm, rotated rx 180 ry 0 rz 90 deg; joints [74.211, -18.142, 89.199, 0, 18.944, 74.211]
  MoveL 9961 to (-66.76, 29.51, -19.34) mm, rotated rx 180 ry 0 rz 90 deg; joints [74.157, -18.123, 89.195, 0, 18.928, 74.157]
  MoveL 9962 to (-66.92, 28.01, -19.75) mm, rotated rx 180 ry 0 rz 90 deg; joints [74.105, -18.098, 89.163, 0, 18.935, 74.105]
  MoveL 9963 to (-66.92, 8.05, -19.75) mm, rotated rx -180 ry 0 rz 90 deg; joints [73.433, -18.012, 88.773, 0, 19.239, 73.433]
  MoveL 9964 to (-66.9, 7.58, -19.75) mm, rotated rx -180 ry 0 rz 90 deg; joints [73.417, -18.009, 88.762, 0, 19.247, 73.417]
  MoveC 9965 to (-65.99, 6.28, -19.75) mm, rotated rx -180 ry 0 rz 90 deg; joints [73.382, -17.99, 88.675, 0, 19.315, 73.382] to (-64.44, 5.94, -19.75) mm, rotated rx 180 ry 0 rz 90 deg; joints [73.386, -17.965, 88.564, 0, 19.401, 73.386]
  MoveL 9966 to (-63.97, 6.05, -19.75) mm, rotated rx 180 ry 0 rz 90 deg; joints [73.395, -17.958, 88.534, 0, 19.424, 73.395]
  MoveL 9967 to (-56.39, 8, -19.75) mm, rotated rx -180 ry 0 rz 90 deg; joints [73.536, -17.851, 88.061, 0, 19.79, 73.536]
  MoveL 9968 to (-54.62, 8.46, -19.75) mm, rotated rx -180 ry 0 rz 90 deg; joints [73.568, -17.826, 87.951, 0, 19.875, 73.568]
  MoveL 9969 to (-54.62, 43.7, -19.75) mm, rotated rx -180 ry 0 rz 90 deg; joints [74.751, -17.979, 88.629, 0, 19.351, 74.751]
  MoveL 9970 to (-63.62, 49.75, -19.75) mm, rotated rx 180 ry 0 rz 90 deg; joints [74.873, -18.139, 89.347, 0, 18.791, 74.873]
  MoveL 9971 to (-63.97, 49.91, -19.75) mm, rotated rx -180 ry 0 rz 90 deg; joints [74.875, -18.144, 89.373, 0, 18.771, 74.875]
  MoveL 9972 to (-64.25, 49.94, -19.75) mm, rotated rx 180 ry 0 rz 90 deg; joints [74.874, -18.148, 89.393, 0, 18.756, 74.874]
  MoveC 9973 to (-65.82, 49.61, -19.75) mm, rotated rx 180 ry 0 rz 90 deg; joints [74.848, -18.17, 89.492, 0, 18.678, 74.848] to (-66.91, 48.43, -19.75) mm, rotated rx -180 ry 0 rz 90 deg; joints [74.798, -18.182, 89.544, 0, 18.637, 74.798]
  MoveL 9974 to (-66.92, 48.33, -19.75) mm, rotated rx -180 ry 0 rz 90 deg; joints [74.794, -18.181, 89.543, 0, 18.639, 74.794]
  MoveL 9975 to (-66.92, 28.01, -19.75) mm, rotated rx 180 ry 0 rz 90 deg; joints [74.105, -18.098, 89.163, 0, 18.935, 74.105]
  MoveL 9976 to (-59.37, 28.01, -19.75) mm, rotated rx 180 ry 0 rz 90 deg; joints [74.177, -17.985, 88.655, 0, 19.33, 74.177]
  MoveL 9977 to (-59.37, 28.01, -16.75) mm, rotated rx -180 ry 0 rz 90 deg; joints [74.177, -18.142, 88.758, 0, 19.384, 74.177]
  Establecer velocidad (1000.0 mm/s)
  MoveL 9978 to (-59.37, 28.01, 10) mm, rotated rx 180 ry 0 rz 90 deg; joints [74.177, -19.538, 89.66, 0, 19.878, 74.177]
  Establecer velocidad (66.7 mm/s)
  MoveL 9979 to (-66.76, 40.13, 10) mm, rotated rx 180 ry 0 rz 90 deg; joints [74.517, -19.704, 90.386, 0, 19.318, 74.517]
  MoveL 9980 to (-66.76, 40.13, -16.75) mm, rotated rx 180 ry 0 rz 90 deg; joints [74.517, -18.303, 89.484, 0, 18.819, 74.517]
  MoveL 9981 to (-66.75, 28.01, -20) mm, rotated rx -180 ry 0 rz 90 deg; joints [74.107, -18.083, 89.143, 0, 18.939, 74.107]
  MoveL 9982 to (-66.75, 8.05, -20) mm, rotated rx -180 ry 0 rz 90 deg; joints [73.434, -17.996, 88.753, 0, 19.243, 73.434]
  MoveC 9983 to (-66.58, 7.26, -20) mm, rotated rx 180 ry 0 rz 90 deg; joints [73.41, -17.99, 88.725, 0, 19.264, 73.41] to (-66.06, 6.63, -20) mm, rotated rx 180 ry 0 rz 90 deg; joints [73.394, -17.979, 88.678, 0, 19.301, 73.394]
  MoveC 9984 to (-65.18, 6.14, -20) mm, rotated rx 180 ry 0 rz 90 deg; joints [73.386, -17.964, 88.609, 0, 19.355, 73.386] to (-64.16, 6.14, -20) mm, rotated rx -180 ry 0 rz 90 deg; joints [73.396, -17.949, 88.541, 0, 19.408, 73.396]
  MoveL 9985 to (-57.48, 7.86, -20) mm, rotated rx -180 ry 0 rz 90 deg; joints [73.52, -17.854, 88.124, 0, 19.73, 73.52]
  MoveL 9986 to (-57.48, 45.46, -20) mm, rotated rx 180 ry 0 rz 90 deg; joints [74.784, -18.017, 88.846, 0, 19.171, 74.784]
  MoveL 9987 to (-63.68, 49.63, -20) mm, rotated rx 180 ry 0 rz 90 deg; joints [74.868, -18.126, 89.34, 0, 18.786, 74.868]
  MoveC 9988 to (-65.47, 49.47, -20) mm, rotated rx -180 ry 0 rz 90 deg; joints [74.847, -18.152, 89.458, 0, 18.694, 74.847] to (-66.75, 48.21, -20) mm, rotated rx 180 ry 0 rz 90 deg; joints [74.792, -18.165, 89.521, 0, 18.644, 74.792]
  MoveL 9989 to (-66.76, 47.86, -20) mm, rotated rx 180 ry 0 rz 90 deg; joints [74.78, -18.164, 89.514, 0, 18.649, 74.78]
  MoveL 9990 to (-66.75, 28.01, -20) mm, rotated rx -180 ry 0 rz 90 deg; joints [74.107, -18.083, 89.143, 0, 18.939, 74.107]
  MoveL 9991 to (-59.2, 28.01, -20) mm, rotated rx 180 ry 0 rz 90 deg; joints [74.179, -17.97, 88.635, 0, 19.335, 74.179]
  MoveL 9992 to (-59.2, 28.01, -17) mm, rotated rx 180 ry 0 rz 90 deg; joints [74.179, -18.126, 88.739, 0, 19.388, 74.179]
  Establecer velocidad (1000.0 mm/s)
  MoveL 9993 to (-59.2, 28.01, 10) mm, rotated rx -180 ry 0 rz 90 deg; joints [74.179, -19.536, 89.649, 0, 19.887, 74.179]
  Establecer velocidad (66.7 mm/s)
  MoveL 9994 to (-57.48, -62.36, 10) mm, rotated rx 180 ry 0 rz 90 deg; joints [71.204, -19.052, 87.623, 0, 21.429, 71.204]
  MoveL 9995 to (-57.48, -62.36, -16.75) mm, rotated rx -180 ry 0 rz 90 deg; joints [71.204, -17.669, 86.722, 0, 20.947, 71.204]
  MoveL 9996 to (-57.48, -50.23, -20) mm, rotated rx 180 ry 0 rz 90 deg; joints [71.599, -17.566, 86.887, 0, 20.68, 71.599]
  MoveL 9997 to (-57.48, -33.76, -20) mm, rotated rx 180 ry 0 rz 90 deg; joints [72.14, -17.653, 87.253, 0, 20.4, 72.14]
  MoveL 9998 to (-58.28, -33.9, -20) mm, rotated rx 180 ry 0 rz 90 deg; joints [72.127, -17.665, 87.304, 0, 20.361, 72.127]
  MoveL 9999 to (-65.14, -35.18, -20) mm, rotated rx 180 ry 0 rz 90 deg; joints [72.011, -17.766, 87.739, 0, 20.027, 72.011]
  MoveC 10000 to (-66.3, -35.86, -20) mm, rotated rx -180 ry 0 rz 90 deg; joints [71.976, -17.78, 87.803, 0, 19.978, 71.976] to (-66.76, -37.13, -20) mm, rotated rx 180 ry 0 rz 90 deg; joints [71.93, -17.781, 87.806, 0, 19.976, 71.93]
  MoveL 10001 to (-66.76, -63.97, -20) mm, rotated rx -180 ry 0 rz 90 deg; joints [71.048, -17.64, 87.2, 0, 20.44, 71.048]
  MoveL 10002 to (-66.75, -64.97, -20) mm, rotated rx 180 ry 0 rz 90 deg; joints [71.015, -17.635, 87.177, 0, 20.458, 71.015]
  MoveC 10003 to (-66.16, -66.37, -20) mm, rotated rx -180 ry 0 rz 90 deg; joints [70.976, -17.618, 87.104, 0, 20.514, 70.976] to (-64.74, -66.94, -20) mm, rotated rx -180 ry 0 rz 90 deg; joints [70.973, -17.592, 86.995, 0, 20.597, 70.973]
  MoveL 10004 to (-63.97, -66.93, -20) mm, rotated rx -180 ry 0 rz 90 deg; joints [70.982, -17.58, 86.943, 0, 20.637, 70.982]
  MoveL 10005 to (-57.48, -66.7, -20) mm, rotated rx -180 ry 0 rz 90 deg; joints [71.062, -17.476, 86.509, 0, 20.967, 71.062]
  MoveL 10006 to (-57.48, -50.23, -20) mm, rotated rx 180 ry 0 rz 90 deg; joints [71.599, -17.566, 86.887, 0, 20.68, 71.599]
  MoveL 10007 to (-65.03, -50.23, -20) mm, rotated rx 180 ry 0 rz 90 deg; joints [71.517, -17.687, 87.398, 0, 20.289, 71.517]
  MoveL 10008 to (-65.03, -50.23, -17) mm, rotated rx 180 ry 0 rz 90 deg; joints [71.517, -17.842, 87.501, 0, 20.341, 71.517]
  Establecer velocidad (1000.0 mm/s)
  MoveL 10009 to (-65.03, -50.23, 10) mm, rotated rx -180 ry 0 rz 90 deg; joints [71.517, -19.244, 88.411, 0, 20.833, 71.517]
  Establecer velocidad (66.7 mm/s)
  MoveL 10010 to (-60.34, -62.36, 10) mm, rotated rx -180 ry 0 rz 90 deg; joints [71.172, -19.1, 87.817, 0, 21.283, 71.172]
  MoveL 10011 to (-60.34, -62.36, -17) mm, rotated rx -180 ry 0 rz 90 deg; joints [71.172, -17.702, 86.907, 0, 20.795, 71.172]
  MoveL 10012 to (-60.34, -50.23, -20.25) mm, rotated rx -180 ry 0 rz 90 deg; joints [71.568, -17.599, 87.072, 0, 20.527, 71.568]
  MoveL 10013 to (-60.34, -34.44, -20.25) mm, rotated rx -180 ry 0 rz 90 deg; joints [72.087, -17.681, 87.423, 0, 20.259, 72.087]
  MoveL 10014 to (-65, -35.31, -20.25) mm, rotated rx 180 ry 0 rz 90 deg; joints [72.009, -17.75, 87.719, 0, 20.031, 72.009]
  MoveC 10015 to (-66.14, -35.98, -20.25) mm, rotated rx 180 ry 0 rz 90 deg; joints [71.974, -17.765, 87.781, 0, 19.984, 71.974] to (-66.59, -37.22, -20.25) mm, rotated rx -180 ry 0 rz 90 deg; joints [71.928, -17.765, 87.784, 0, 19.981, 71.928]
  MoveL 10016 to (-66.59, -63.97, -20.25) mm, rotated rx 180 ry 0 rz 90 deg; joints [71.049, -17.625, 87.18, 0, 20.444, 71.049]
  MoveL 10017 to (-66.59, -64.91, -20.25) mm, rotated rx 180 ry 0 rz 90 deg; joints [71.019, -17.62, 87.158, 0, 20.461, 71.019]
  MoveC 10018 to (-66.08, -66.15, -20.25) mm, rotated rx -180 ry 0 rz 90 deg; joints [70.984, -17.605, 87.095, 0, 20.509, 70.984] to (-64.91, -66.79, -20.25) mm, rotated rx -180 ry 0 rz 90 deg; joints [70.976, -17.583, 87.002, 0, 20.581, 70.976]
  MoveC 10019 to (-62.63, -66.75, -20.25) mm, rotated rx 180 ry 0 rz 90 deg; joints [71.003, -17.546, 86.848, 0, 20.698, 71.003] to (-60.34, -66.66, -20.25) mm, rotated rx -180 ry 0 rz 90 deg; joints [71.032, -17.51, 86.695, 0, 20.815, 71.032]
  MoveL 10020 to (-60.34, -50.23, -20.25) mm, rotated rx -180 ry 0 rz 90 deg; joints [71.568, -17.599, 87.072, 0, 20.527, 71.568]
  MoveL 10021 to (-61, -42.71, -20.25) mm, rotated rx -180 ry 0 rz 90 deg; joints [71.808, -17.649, 87.285, 0, 20.364, 71.808]
  MoveL 10022 to (-61, -42.71, -17.25) mm, rotated rx 180 ry 0 rz 90 deg; joints [71.808, -17.805, 87.388, 0, 20.417, 71.808]
  Establecer velocidad (1000.0 mm/s)
  MoveL 10023 to (-61, -42.71, 10) mm, rotated rx 180 ry 0 rz 90 deg; joints [71.808, -19.219, 88.307, 0, 20.912, 71.808]
  Establecer velocidad (66.7 mm/s)
  MoveL 10024 to (-66.59, 40.15, 10) mm, rotated rx 180 ry 0 rz 90 deg; joints [74.519, -19.702, 90.375, 0, 19.326, 74.519]
  MoveL 10025 to (-66.59, 40.15, -17) mm, rotated rx 180 ry 0 rz 90 deg; joints [74.519, -18.288, 89.465, 0, 18.823, 74.519]
  MoveL 10026 to (-66.59, 28.02, -20.25) mm, rotated rx 180 ry 0 rz 90 deg; joints [74.109, -18.067, 89.124, 0, 18.943, 74.109]
  MoveL 10027 to (-66.59, 9, -20.25) mm, rotated rx 180 ry 0 rz 90 deg; joints [73.468, -17.985, 88.753, 0, 19.232, 73.468]
  MoveL 10028 to (-66.58, 8.05, -20.25) mm, rotated rx -180 ry 0 rz 90 deg; joints [73.436, -17.981, 88.733, 0, 19.247, 73.436]
  MoveC 10029 to (-65.67, 6.6, -20.25) mm, rotated rx -180 ry 0 rz 90 deg; joints [73.396, -17.96, 88.642, 0, 19.318, 73.396] to (-63.97, 6.33, -20.25) mm, rotated rx 180 ry 0 rz 90 deg; joints [73.404, -17.933, 88.523, 0, 19.411, 73.404]
  MoveL 10030 to (-60.34, 7.27, -20.25) mm, rotated rx 180 ry 0 rz 90 deg; joints [73.472, -17.882, 88.297, 0, 19.586, 73.472]
  MoveL 10031 to (-60.34, 47.22, -20.25) mm, rotated rx 180 ry 0 rz 90 deg; joints [74.817, -18.054, 89.063, 0, 18.991, 74.817]
  MoveL 10032 to (-63.49, 49.35, -20.25) mm, rotated rx -180 ry 0 rz 90 deg; joints [74.861, -18.109, 89.314, 0, 18.795, 74.861]
  MoveC 10033 to (-65.29, 49.24, -20.25) mm, rotated rx 180 ry 0 rz 90 deg; joints [74.84, -18.135, 89.433, 0, 18.702, 74.84] to (-66.59, 47.99, -20.25) mm, rotated rx -180 ry 0 rz 90 deg; joints [74.786, -18.149, 89.497, 0, 18.652, 74.786]
  MoveL 10034 to (-66.59, 28.02, -20.25) mm, rotated rx 180 ry 0 rz 90 deg; joints [74.109, -18.067, 89.124, 0, 18.943, 74.109]
  MoveL 10035 to (-65.93, 20.5, -20.25) mm, rotated rx 180 ry 0 rz 90 deg; joints [73.861, -18.025, 88.935, 0, 19.091, 73.861]
  MoveL 10036 to (-65.93, 20.5, -17.25) mm, rotated rx 180 ry 0 rz 90 deg; joints [73.861, -18.182, 89.039, 0, 19.144, 73.861]
  Establecer velocidad (1000.0 mm/s)
  MoveL 10037 to (-65.93, 20.5, 10) mm, rotated rx -180 ry 0 rz 90 deg; joints [73.861, -19.607, 89.957, 0, 19.649, 73.861]
  Establecer velocidad (66.7 mm/s)
  MoveL 10038 to (-66.43, 40.15, 10) mm, rotated rx 180 ry 0 rz 90 deg; joints [74.521, -19.699, 90.364, 0, 19.335, 74.521]
  MoveL 10039 to (-66.43, 40.15, -17.25) mm, rotated rx -180 ry 0 rz 90 deg; joints [74.521, -18.272, 89.445, 0, 18.827, 74.521]
  MoveL 10040 to (-66.43, 28.02, -20.5) mm, rotated rx -180 ry 0 rz 90 deg; joints [74.11, -18.052, 89.104, 0, 18.947, 74.11]
  MoveL 10041 to (-66.43, 9, -20.5) mm, rotated rx -180 ry 0 rz 90 deg; joints [73.469, -17.969, 88.733, 0, 19.236, 73.469]
  MoveL 10042 to (-66.41, 8.05, -20.5) mm, rotated rx 180 ry 0 rz 90 deg; joints [73.438, -17.965, 88.713, 0, 19.252, 73.438]
  MoveC 10043 to (-65.55, 6.8, -20.5) mm, rotated rx 180 ry 0 rz 90 deg; joints [73.404, -17.946, 88.63, 0, 19.316, 73.404] to (-64.06, 6.46, -20.5) mm, rotated rx 180 ry 0 rz 90 deg; joints [73.408, -17.922, 88.523, 0, 19.399, 73.408]
  MoveC 10044 to (-63.63, 6.55, -20.5) mm, rotated rx -180 ry 0 rz 90 deg; joints [73.415, -17.916, 88.495, 0, 19.421, 73.415] to (-63.2, 6.67, -20.5) mm, rotated rx -180 ry 0 rz 90 deg; joints [73.424, -17.91, 88.469, 0, 19.441, 73.424]
  MoveL 10045 to (-63.2, 48.99, -20.5) mm, rotated rx -180 ry 0 rz 90 deg; joints [74.851, -18.09, 89.279, 0, 18.811, 74.851]
  MoveL 10046 to (-63.43, 49.15, -20.5) mm, rotated rx 180 ry 0 rz 90 deg; joints [74.854, -18.094, 89.297, 0, 18.797, 74.854]
  MoveC 10047 to (-65.17, 48.98, -20.5) mm, rotated rx 180 ry 0 rz 90 deg; joints [74.833, -18.119, 89.411, 0, 18.708, 74.833] to (-66.43, 47.76, -20.5) mm, rotated rx 180 ry 0 rz 90 deg; joints [74.78, -18.132, 89.473, 0, 18.659, 74.78]
  MoveL 10048 to (-66.43, 28.02, -20.5) mm, rotated rx -180 ry 0 rz 90 deg; joints [74.11, -18.052, 89.104, 0, 18.947, 74.11]
  MoveL 10049 to (-66.43, 20.47, -20.5) mm, rotated rx 180 ry 0 rz 90 deg; joints [73.855, -18.02, 88.959, 0, 19.061, 73.855]
  MoveL 10050 to (-66.43, 20.47, -17.5) mm, rotated rx 180 ry 0 rz 90 deg; joints [73.855, -18.177, 89.062, 0, 19.114, 73.855]
  Establecer velocidad (1000.0 mm/s)
  MoveL 10051 to (-66.43, 20.47, 10) mm, rotated rx -180 ry 0 rz 90 deg; joints [73.855, -19.614, 89.99, 0, 19.624, 73.855]
  Establecer velocidad (66.7 mm/s)
  MoveL 10052 to (-63.2, -63, 10) mm, rotated rx -180 ry 0 rz 90 deg; joints [71.119, -19.143, 87.995, 0, 21.148, 71.119]
  MoveL 10053 to (-63.2, -63, -17.25) mm, rotated rx 180 ry 0 rz 90 deg; joints [71.119, -17.732, 87.077, 0, 20.655, 71.119]
  MoveL 10054 to (-63.2, -50.87, -20.5) mm, rotated rx 180 ry 0 rz 90 deg; joints [71.516, -17.628, 87.242, 0, 20.386, 71.516]
  MoveL 10055 to (-63.2, -35.12, -20.5) mm, rotated rx 180 ry 0 rz 90 deg; joints [72.034, -17.71, 87.592, 0, 20.118, 72.034]
  MoveL 10056 to (-64.86, -35.43, -20.5) mm, rotated rx 180 ry 0 rz 90 deg; joints [72.006, -17.734, 87.698, 0, 20.037, 72.006]
  MoveC 10057 to (-65.98, -36.09, -20.5) mm, rotated rx -180 ry 0 rz 90 deg; joints [71.972, -17.748, 87.759, 0, 19.989, 71.972] to (-66.43, -37.32, -20.5) mm, rotated rx 180 ry 0 rz 90 deg; joints [71.927, -17.749, 87.762, 0, 19.987, 71.927]
  MoveL 10058 to (-66.43, -63.97, -20.5) mm, rotated rx 180 ry 0 rz 90 deg; joints [71.051, -17.609, 87.161, 0, 20.449, 71.051]
  MoveL 10059 to (-66.42, -64.75, -20.5) mm, rotated rx -180 ry 0 rz 90 deg; joints [71.026, -17.605, 87.142, 0, 20.463, 71.026]
  MoveC 10060 to (-65.89, -66.05, -20.5) mm, rotated rx -180 ry 0 rz 90 deg; joints [70.989, -17.589, 87.076, 0, 20.513, 70.989] to (-64.62, -66.63, -20.5) mm, rotated rx 180 ry 0 rz 90 deg; joints [70.985, -17.566, 86.976, 0, 20.589, 70.985]
  MoveC 10061 to (-63.9, -66.65, -20.5) mm, rotated rx 180 ry 0 rz 90 deg; joints [70.992, -17.554, 86.928, 0, 20.626, 70.992] to (-63.2, -66.62, -20.5) mm, rotated rx 180 ry 0 rz 90 deg; joints [71.001, -17.543, 86.881, 0, 20.662, 71.001]
  MoveL 10062 to (-63.2, -50.87, -20.5) mm, rotated rx 180 ry 0 rz 90 deg; joints [71.516, -17.628, 87.242, 0, 20.386, 71.516]
  MoveL 10063 to (-63.2, -43.32, -20.5) mm, rotated rx 180 ry 0 rz 90 deg; joints [71.764, -17.668, 87.411, 0, 20.257, 71.764]
  MoveL 10064 to (-63.2, -43.32, -17.5) mm, rotated rx 180 ry 0 rz 90 deg; joints [71.764, -17.824, 87.515, 0, 20.309, 71.764]
  Establecer velocidad (1000.0 mm/s)
  MoveL 10065 to (-63.2, -43.32, 10) mm, rotated rx -180 ry 0 rz 90 deg; joints [71.764, -19.251, 88.442, 0, 20.809, 71.764]
  Establecer velocidad (66.7 mm/s)
  MoveL 10066 to (-66.05, -63, 10) mm, rotated rx 180 ry 0 rz 90 deg; joints [71.087, -19.19, 88.188, 0, 21.002, 71.087]
  MoveL 10067 to (-66.05, -63, -17.5) mm, rotated rx -180 ry 0 rz 90 deg; joints [71.087, -17.764, 87.261, 0, 20.503, 71.087]
  MoveL 10068 to (-66.05, -50.87, -20.75) mm, rotated rx -180 ry 0 rz 90 deg; joints [71.485, -17.66, 87.426, 0, 20.234, 71.485]
  MoveL 10069 to (-66.05, -36.52, -20.75) mm, rotated rx 180 ry 0 rz 90 deg; joints [71.957, -17.734, 87.746, 0, 19.989, 71.957]
  MoveC 10070 to (-66.21, -36.96, -20.75) mm, rotated rx -180 ry 0 rz 90 deg; joints [71.941, -17.735, 87.747, 0, 19.988, 71.941] to (-66.26, -37.43, -20.75) mm, rotated rx -180 ry 0 rz 90 deg; joints [71.925, -17.733, 87.74, 0, 19.993, 71.925]
  MoveL 10071 to (-66.26, -64.73, -20.75) mm, rotated rx -180 ry 0 rz 90 deg; joints [71.028, -17.589, 87.123, 0, 20.466, 71.028]
  MoveC 10072 to (-66.21, -65.12, -20.75) mm, rotated rx -180 ry 0 rz 90 deg; joints [71.016, -17.586, 87.111, 0, 20.476, 71.016] to (-66.05, -65.48, -20.75) mm, rotated rx 180 ry 0 rz 90 deg; joints [71.006, -17.582, 87.092, 0, 20.49, 71.006]
  MoveL 10073 to (-66.05, -50.87, -20.75) mm, rotated rx -180 ry 0 rz 90 deg; joints [71.485, -17.66, 87.426, 0, 20.234, 71.485]
  MoveL 10074 to (-66.05, -50.87, -17.75) mm, rotated rx 180 ry 0 rz 90 deg; joints [71.485, -17.816, 87.53, 0, 20.286, 71.485]
  Establecer velocidad (1000.0 mm/s)
  MoveL 10075 to (-66.05, -50.87, 10) mm, rotated rx 180 ry 0 rz 90 deg; joints [71.485, -19.257, 88.465, 0, 20.791, 71.485]
  Establecer velocidad (66.7 mm/s)
  MoveL 10076 to (-66.05, 15.67, 10) mm, rotated rx 180 ry 0 rz 90 deg; joints [73.697, -19.587, 89.871, 0, 19.716, 73.697]
  MoveL 10077 to (-66.05, 15.67, -17.5) mm, rotated rx 180 ry 0 rz 90 deg; joints [73.697, -18.15, 88.943, 0, 19.207, 73.697]
  MoveL 10078 to (-66.05, 27.8, -20.75) mm, rotated rx -180 ry 0 rz 90 deg; joints [74.106, -18.032, 89.066, 0, 18.966, 74.106]
  MoveL 10079 to (-66.05, 47.94, -20.75) mm, rotated rx 180 ry 0 rz 90 deg; joints [74.789, -18.115, 89.443, 0, 18.672, 74.789]
  MoveL 10080 to (-66.26, 47.55, -20.75) mm, rotated rx -180 ry 0 rz 90 deg; joints [74.774, -18.116, 89.45, 0, 18.666, 74.774]
  MoveL 10081 to (-66.26, 8.42, -20.75) mm, rotated rx -180 ry 0 rz 90 deg; joints [73.452, -17.951, 88.702, 0, 19.25, 73.452]
  MoveC 10082 to (-66.21, 8.02, -20.75) mm, rotated rx -180 ry 0 rz 90 deg; joints [73.439, -17.949, 88.69, 0, 19.259, 73.439] to (-66.05, 7.65, -20.75) mm, rotated rx 180 ry 0 rz 90 deg; joints [73.428, -17.945, 88.672, 0, 19.273, 73.428]
  MoveL 10083 to (-66.05, 27.8, -20.75) mm, rotated rx -180 ry 0 rz 90 deg; joints [74.106, -18.032, 89.066, 0, 18.966, 74.106]
  MoveL 10084 to (-66.05, 27.8, -17.75) mm, rotated rx -180 ry 0 rz 90 deg; joints [74.106, -18.189, 89.17, 0, 19.019, 74.106]
  Establecer velocidad (1000.0 mm/s)
  MoveL 10085 to (-66.05, 27.8, 10) mm, rotated rx 180 ry 0 rz 90 deg; joints [74.106, -19.641, 90.106, 0, 19.534, 74.106]
  MoveL 10086 to (-66.05, 27.8, 10) mm, rotated rx 180 ry 0 rz 90 deg; joints [74.106, -19.641, 90.106, 0, 19.534, 74.106]
  MoveL 10087 to (-66.05, 27.8, 110) mm, rotated rx 180 ry 0 rz 90 deg; joints [74.106, -24.845, 93.138, 0, 21.707, 74.106]
